// TwinCAT 3 PLC project TcSpeech_Sample_Eventlogger
// ProgramVersion: 3.1.4026.9
// libraries:
//   Tc2_Standard, * (Beckhoff Automation GmbH)
//   Tc2_System, * (Beckhoff Automation GmbH)
//   Tc3_EventLogger, * (Beckhoff Automation GmbH)
//   Tc3_Speech, * (Beckhoff Automation GmbH)
// project tree:
//   / PlcTask.TcTTO
//   POUs/ MAIN.TcPOU
// real-time tasks:
//   TASK PlcTask: cycle T#10ms, priority 20, ADS port 350

CONFIGURATION TcSpeech_Sample_Eventlogger
    RESOURCE PLC ON TwinCAT3
        TASK PlcTask(INTERVAL := T#10ms, PRIORITY := 20);
        PROGRAM MAIN WITH PlcTask : MAIN;
    END_RESOURCE
END_CONFIGURATION

// ---- POUs/MAIN.TcPOU
// TwinCAT Speech Eventlogger Sample
// Event-To-Speech: If "EventSpeechTestClass.TTSEvent" is detected by TcSpeech Service, it will be synthesised
// Speech-To-Event: If "Hello TwinCAT" is recognized, the "EventSpeechTestClass.ASREvent" will be sent by TcSpeech (see LoggedEvents-Window)
PROGRAM MAIN
VAR
	fbEvent 	: FB_TcEventLogger; 
	bSendEvent	: BOOL;
END_VAR

// Event-To-Speech: Set bSendEvent to true, to send event and listen for output
IF bSendEvent THEN 
	fbEvent.SendMessageEx(TC_EVENTS.EventSpeechTestClass.TTSEvent, 0, 0, 0);
	bSendEvent := FALSE; 
END_IF

// Speech-to-Event: 
// Speech Recognition will be started automatically by TcSpeech Service, no more PLC code necessary

END_PROGRAM
